    LOCAL CONST Robtarget Tr_meulage_bavure_379 := [[8.9303857421875,-168.09725,77.5905703125],[0.760092273440949,-0.627413460069246,0.107679305140414,-0.130450194418344],[0,0,0,0],[8.999999E+09,8.999999E+09,8.999999E+09,8.999999E+09,8.999999E+09,8.999999E+09]];
    LOCAL CONST Robtarget Tr_meulage_bavure_380 := [[6.36778564453125,-166.2545,77.61740625],[0.757380069640721,-0.624678423253224,0.120981857756658,-0.146682267935255],[0,0,0,0],[8.999999E+09,8.999999E+09,8.999999E+09,8.999999E+09,8.999999E+09,8.999999E+09]];
    LOCAL CONST Robtarget Tr_meulage_bavure_381 := [[0.0211522235870361,-161.8668125,77.659015625],[0.755787418378999,-0.622904489845863,0.128428166406746,-0.155825481944626],[0,0,0,0],[8.999999E+09,8.999999E+09,8.999999E+09,8.999999E+09,8.999999E+09,8.999999E+09]];
    LOCAL CONST Robtarget Tr_meulage_bavure_382 := [[-4.13824365234375,-159.009953125,77.6836484375],[0.75532643398599,-0.622107777939022,0.131008038074695,-0.159062203900237],[0,0,0,0],[8.999999E+09,8.999999E+09,8.999999E+09,8.999999E+09,8.999999E+09,8.999999E+09]];
    LOCAL CONST Robtarget Tr_meulage_bavure_383 := [[-6.49300439453125,-157.311875,77.7089765625],[0.755817096690397,-0.622133912444517,0.129761641555208,-0.157644624766832],[0,0,0,0],[8.999999E+09,8.999999E+09,8.999999E+09,8.999999E+09,8.999999E+09,8.999999E+09]];
    LOCAL CONST Robtarget Tr_meulage_bavure_384 := [[-7.27819287109375,-156.766953125,77.714421875],[0.756985671882866,-0.622757763981476,0.125698769882492,-0.152791620237717],[0,0,0,0],[8.999999E+09,8.999999E+09,8.999999E+09,8.999999E+09,8.999999E+09,8.999999E+09]];
    LOCAL CONST Robtarget Tr_meulage_bavure_385 := [[-7.3110322265625,-156.78715625,77.7085859375],[0.758538176477072,-0.623736548693659,0.119790927466895,-0.14568008219102],[0,0,0,0],[8.999999E+09,8.999999E+09,8.999999E+09,8.999999E+09,8.999999E+09,8.999999E+09]];
    LOCAL CONST Robtarget Tr_meulage_bavure_386 := [[-10.1234833984375,-155.486203125,77.6362265625],[0.760196318256337,-0.624846439022857,0.112999081170998,-0.137476154312211],[0,0,0,0],[8.999999E+09,8.999999E+09,8.999999E+09,8.999999E+09,8.999999E+09,8.999999E+09]];
    LOCAL CONST Robtarget Tr_meulage_bavure_387 := [[-10.6625419921875,-155.202578125,77.6271875],[0.761746908687365,-0.625914144918721,0.106180842065471,-0.129223678457846],[0,0,0,0],[8.999999E+09,8.999999E+09,8.999999E+09,8.999999E+09,8.999999E+09,8.999999E+09]];
    LOCAL CONST Robtarget Tr_meulage_bavure_388 := [[-12.2218876953125,-154.823703125,77.53875],[0.763048486638023,-0.626818658409292,0.100073150713779,-0.121822580072891],[0,0,0,0],[8.999999E+09,8.999999E+09,8.999999E+09,8.999999E+09,8.999999E+09,8.999999E+09]];
    LOCAL CONST Robtarget Tr_meulage_bavure_389 := [[-13.7799794921875,-154.60521875,77.42778125],[0.764015045491845,-0.62749443057358,0.0952699651388726,-0.115997343088844],[0,0,0,0],[8.999999E+09,8.999999E+09,8.999999E+09,8.999999E+09,8.999999E+09,8.999999E+09]];
    LOCAL CONST Robtarget Tr_meulage_bavure_390 := [[-14.96165625,-154.561921875,77.3263515625],[0.764604259131724,-0.627907931444273,0.0922133285385718,-0.112288283390735],[0,0,0,0],[8.999999E+09,8.999999E+09,8.999999E+09,8.999999E+09,8.999999E+09,8.999999E+09]];
    LOCAL CONST Robtarget Tr_meulage_bavure_391 := [[-16.279068359375,-154.44878125,77.222421875],[0.764800293575778,-0.62804670288681,0.0911701159971482,-0.111021889231259],[0,0,0,0],[8.999999E+09,8.999999E+09,8.999999E+09,8.999999E+09,8.999999E+09,8.999999E+09]];
    !
    !Declaration des points de tronconnage

    !
    !Cycle
    LOCAL PROC Cycle()
        !
        Prise;
        !
        Meulage;
        !
        !
        Depose;
        !
    ENDPROC

    !Trajectoire de prise de la pièce
    LOCAL PROC PRISE()

		!
        !Trigger localisation
        LocalisationPieceTable 810 \model:=1;
        !
        !Approche
		MoveJ Reltool(PicKPosition,0,0,-100),V1000,Z0,Tool_Prehenseur1 \Wobj:=Wobj_vision;
		MoveL Reltool(PicKPosition,0,0,-50),V500,Z0,Tool_Prehenseur1 \Wobj:=Wobj_vision;
		MoveL Reltool(PicKPosition,0,0,-10),V200,Z0,Tool_Prehenseur1 \Wobj:=Wobj_vision;
		MoveL PicKPosition,V100,Fine,Tool_Prehenseur1 \Wobj:=Wobj_vision;

        !Fermeture pince
		Gripper_Close;
        !
		MoveL Reltool(PicKPosition,0,0,-100),V500,Z0,Tool_Prehenseur1 \Wobj:=Wobj_vision;

        !Trigger relocalisation
		LocalisationPiecePrehenseur 810 \model:=1,Ref;
        !
        PEO;
        !
    ENDPROC

    !Trajectoire de tronconnage
    LOCAL PROC Tronconnage()
        !
        !StartMotor1();
        !
        ConfJ \Off;
        ConfL \Off;


    ENDPROC


    !Trajectoire de meulage
    LOCAL PROC Meulage()
        !
        !StartMotor2();
        !

        ConfJ \Off;
        ConfL \Off;


        !---------- Meulage zone : 1 ------------

        !Approche PLAN

        Go_to_Meulage_Plan;
		Tool := ToolOffset(Tool_M1_D500_S0 \Z);

        !
        !Approche
        MoveJ Reltool(Tr_meulage_motif_1_0,0,0,-200),V1000,Z0,Tool \Wobj:=Wobj_Part_0;
        MoveL Reltool(Tr_meulage_motif_1_0,0,0,-100),V500,Z0,Tool \Wobj:=Wobj_Part_0;
        MoveL Reltool(Tr_meulage_motif_1_0,0,0,-10),V100,Z0,Tool \Wobj:=Wobj_Part_0;
        !
        !Trajectoire
        Movel Tr_meulage_motif_1_0,VitesseLente,Z0,Tool \Wobj:=Wobj_Part_0;
        Movel Tr_meulage_motif_1_1,VitesseLente,Z0,Tool \Wobj:=Wobj_Part_0;
        Movel Tr_meulage_motif_1_2,VitesseLente,Z0,Tool \Wobj:=Wobj_Part_0;
        Movel Tr_meulage_motif_1_3,VitesseLente,Z0,Tool \Wobj:=Wobj_Part_0;
        Movel Tr_meulage_motif_1_4,VitesseLente,Z0,Tool \Wobj:=Wobj_Part_0;
        Movel Tr_meulage_motif_1_5,VitesseLente,Z0,Tool \Wobj:=Wobj_Part_0;
        Movel Tr_meulage_motif_1_6,VitesseLente,Z0,Tool \Wobj:=Wobj_Part_0;
        Movel Tr_meulage_motif_1_7,VitesseLente,Z0,Tool \Wobj:=Wobj_Part_0;
        Movel Tr_meulage_motif_1_8,VitesseLente,Z0,Tool \Wobj:=Wobj_Part_0;
        Movel Tr_meulage_motif_1_9,VitesseLente,Z0,Tool \Wobj:=Wobj_Part_0;
        Movel Tr_meulage_motif_1_10,VitesseLente,Z0,Tool \Wobj:=Wobj_Part_0;
        Movel Tr_meulage_motif_1_11,VitesseLente,Z0,Tool \Wobj:=Wobj_Part_0;
        Movel Tr_meulage_motif_1_12,VitesseLente,Z0,Tool \Wobj:=Wobj_Part_0;
        Movel Tr_meulage_motif_1_13,VitesseLente,Z0,Tool \Wobj:=Wobj_Part_0;
        Movel Tr_meulage_motif_1_14,VitesseLente,Z0,Tool \Wobj:=Wobj_Part_0;
        Movel Tr_meulage_motif_1_15,VitesseLente,Z0,Tool \Wobj:=Wobj_Part_0;
        Movel Tr_meulage_motif_1_16,VitesseLente,Z0,Tool \Wobj:=Wobj_Part_0;
        Movel Tr_meulage_motif_1_17,VitesseLente,Z0,Tool \Wobj:=Wobj_Part_0;
        Movel Tr_meulage_motif_1_18,VitesseLente,Z0,Tool \Wobj:=Wobj_Part_0;
        Movel Tr_meulage_motif_1_19,VitesseLente,Z0,Tool \Wobj:=Wobj_Part_0;
        Movel Tr_meulage_motif_1_20,VitesseLente,Z0,Tool \Wobj:=Wobj_Part_0;
        Movel Tr_meulage_motif_1_21,VitesseLente,Z0,Tool \Wobj:=Wobj_Part_0;
        Movel Tr_meulage_motif_1_22,VitesseLente,Z0,Tool \Wobj:=Wobj_Part_0;
        Movel Tr_meulage_motif_1_23,VitesseLente,Z0,Tool \Wobj:=Wobj_Part_0;
        Movel Tr_meulage_motif_1_24,VitesseLente,Z0,Tool \Wobj:=Wobj_Part_0;
        Movel Tr_meulage_motif_1_25,VitesseLente,Z0,Tool \Wobj:=Wobj_Part_0;
        Movel Tr_meulage_motif_1_26,VitesseLente,Z0,Tool \Wobj:=Wobj_Part_0;
        Movel Tr_meulage_motif_1_27,VitesseLente,Z0,Tool \Wobj:=Wobj_Part_0;
        Movel Tr_meulage_motif_1_28,VitesseLente,Z0,Tool \Wobj:=Wobj_Part_0;
        Movel Tr_meulage_motif_1_29,VitesseLente,Z0,Tool \Wobj:=Wobj_Part_0;
        Movel Tr_meulage_motif_1_30,VitesseLente,Z0,Tool \Wobj:=Wobj_Part_0;
        Movel Tr_meulage_motif_1_31,VitesseLente,Z0,Tool \Wobj:=Wobj_Part_0;
        Movel Tr_meulage_motif_1_32,VitesseLente,Z0,Tool \Wobj:=Wobj_Part_0;
        Movel Tr_meulage_motif_1_33,VitesseLente,Z0,Tool \Wobj:=Wobj_Part_0;
        Movel Tr_meulage_motif_1_34,VitesseLente,Z0,Tool \Wobj:=Wobj_Part_0;
        Movel Tr_meulage_motif_1_35,VitesseLente,Z0,Tool \Wobj:=Wobj_Part_0;
        Movel Tr_meulage_motif_1_36,VitesseLente,Z0,Tool \Wobj:=Wobj_Part_0;
        Movel Tr_meulage_motif_1_37,VitesseLente,Z0,Tool \Wobj:=Wobj_Part_0;
        Movel Tr_meulage_motif_1_38,VitesseLente,Z0,Tool \Wobj:=Wobj_Part_0;
        Movel Tr_meulage_motif_1_39,VitesseLente,Z0,Tool \Wobj:=Wobj_Part_0;
        Movel Tr_meulage_motif_1_40,VitesseLente,Z0,Tool \Wobj:=Wobj_Part_0;
        Movel Tr_meulage_motif_1_41,VitesseLente,Z0,Tool \Wobj:=Wobj_Part_0;
        Movel Tr_meulage_motif_1_42,VitesseLente,Z0,Tool \Wobj:=Wobj_Part_0;
        Movel Tr_meulage_motif_1_43,VitesseLente,Z0,Tool \Wobj:=Wobj_Part_0;
        Movel Tr_meulage_motif_1_44,VitesseLente,Z0,Tool \Wobj:=Wobj_Part_0;
        Movel Tr_meulage_motif_1_45,VitesseLente,Z0,Tool \Wobj:=Wobj_Part_0;
        Movel Tr_meulage_motif_1_46,VitesseLente,Z0,Tool \Wobj:=Wobj_Part_0;
        Movel Tr_meulage_motif_1_47,VitesseLente,Z0,Tool \Wobj:=Wobj_Part_0;
        Movel Tr_meulage_motif_1_48,VitesseLente,Z0,Tool \Wobj:=Wobj_Part_0;
        Movel Tr_meulage_motif_1_49,VitesseLente,Z0,Tool \Wobj:=Wobj_Part_0;
        Movel Tr_meulage_motif_1_50,VitesseLente,Z0,Tool \Wobj:=Wobj_Part_0;
        Movel Tr_meulage_motif_1_51,VitesseLente,Z0,Tool \Wobj:=Wobj_Part_0;
        Movel Tr_meulage_motif_1_52,VitesseLente,Z0,Tool \Wobj:=Wobj_Part_0;
        Movel Tr_meulage_motif_1_53,VitesseLente,Z0,Tool \Wobj:=Wobj_Part_0;
        Movel Tr_meulage_motif_1_54,VitesseLente,Z0,Tool \Wobj:=Wobj_Part_0;
        Movel Tr_meulage_motif_1_55,VitesseLente,Z0,Tool \Wobj:=Wobj_Part_0;
        Movel Tr_meulage_motif_1_56,VitesseLente,Z0,Tool \Wobj:=Wobj_Part_0;
        Movel Tr_meulage_motif_1_57,VitesseLente,Z0,Tool \Wobj:=Wobj_Part_0;
        Movel Tr_meulage_motif_1_58,VitesseLente,Z0,Tool \Wobj:=Wobj_Part_0;
        Movel Tr_meulage_motif_1_59,VitesseLente,Z0,Tool \Wobj:=Wobj_Part_0;
        Movel Tr_meulage_motif_1_60,VitesseLente,Z0,Tool \Wobj:=Wobj_Part_0;
        Movel Tr_meulage_motif_1_61,VitesseLente,Z0,Tool \Wobj:=Wobj_Part_0;
        Movel Tr_meulage_motif_1_62,VitesseLente,Z0,Tool \Wobj:=Wobj_Part_0;
        Movel Tr_meulage_motif_1_63,VitesseLente,Z0,Tool \Wobj:=Wobj_Part_0;
        Movel Tr_meulage_motif_1_64,VitesseLente,Z0,Tool \Wobj:=Wobj_Part_0;
        Movel Tr_meulage_motif_1_65,VitesseLente,Z0,Tool \Wobj:=Wobj_Part_0;
        Movel Tr_meulage_motif_1_66,VitesseLente,Z0,Tool \Wobj:=Wobj_Part_0;
        Movel Tr_meulage_motif_1_67,VitesseLente,Z0,Tool \Wobj:=Wobj_Part_0;
        Movel Tr_meulage_motif_1_68,VitesseLente,Z0,Tool \Wobj:=Wobj_Part_0;
        Movel Tr_meulage_motif_1_69,VitesseLente,Z0,Tool \Wobj:=Wobj_Part_0;
        Movel Tr_meulage_motif_1_70,VitesseLente,Z0,Tool \Wobj:=Wobj_Part_0;
        Movel Tr_meulage_motif_1_71,VitesseLente,Z0,Tool \Wobj:=Wobj_Part_0;
        Movel Tr_meulage_motif_1_72,VitesseLente,Z0,Tool \Wobj:=Wobj_Part_0;
        Movel Tr_meulage_motif_1_73,VitesseLente,Z0,Tool \Wobj:=Wobj_Part_0;
        Movel Tr_meulage_motif_1_74,VitesseLente,Z0,Tool \Wobj:=Wobj_Part_0;
        Movel Tr_meulage_motif_1_75,VitesseLente,Z0,Tool \Wobj:=Wobj_Part_0;
        Movel Tr_meulage_motif_1_76,VitesseLente,Z0,Tool \Wobj:=Wobj_Part_0;
        Movel Tr_meulage_motif_1_77,VitesseLente,Z0,Tool \Wobj:=Wobj_Part_0;
        Movel Tr_meulage_motif_1_78,VitesseLente,Z0,Tool \Wobj:=Wobj_Part_0;
        Movel Tr_meulage_motif_1_79,VitesseLente,Z0,Tool \Wobj:=Wobj_Part_0;
        Movel Tr_meulage_motif_1_80,VitesseLente,Z0,Tool \Wobj:=Wobj_Part_0;
        Movel Tr_meulage_motif_1_81,VitesseLente,Z0,Tool \Wobj:=Wobj_Part_0;
        Movel Tr_meulage_motif_1_82,VitesseLente,Z0,Tool \Wobj:=Wobj_Part_0;
        Movel Tr_meulage_motif_1_83,VitesseLente,Z0,Tool \Wobj:=Wobj_Part_0;
        Movel Tr_meulage_motif_1_84,VitesseLente,Z0,Tool \Wobj:=Wobj_Part_0;
        Movel Tr_meulage_motif_1_85,VitesseLente,Z0,Tool \Wobj:=Wobj_Part_0;
        Movel Tr_meulage_motif_1_86,VitesseLente,Z0,Tool \Wobj:=Wobj_Part_0;
        Movel Tr_meulage_motif_1_87,VitesseLente,Z0,Tool \Wobj:=Wobj_Part_0;
        Movel Tr_meulage_motif_1_88,VitesseLente,Z0,Tool \Wobj:=Wobj_Part_0;
        Movel Tr_meulage_motif_1_89,VitesseLente,Z0,Tool \Wobj:=Wobj_Part_0;
        Movel Tr_meulage_motif_1_90,VitesseLente,Z0,Tool \Wobj:=Wobj_Part_0;
        Movel Tr_meulage_motif_1_91,VitesseLente,Z0,Tool \Wobj:=Wobj_Part_0;
        Movel Tr_meulage_motif_1_92,VitesseLente,Z0,Tool \Wobj:=Wobj_Part_0;
        Movel Tr_meulage_motif_1_93,VitesseLente,Z0,Tool \Wobj:=Wobj_Part_0;
        Movel Tr_meulage_motif_1_94,VitesseLente,Z0,Tool \Wobj:=Wobj_Part_0;
        Movel Tr_meulage_motif_1_95,VitesseLente,Z0,Tool \Wobj:=Wobj_Part_0;
        Movel Tr_meulage_motif_1_96,VitesseLente,Z0,Tool \Wobj:=Wobj_Part_0;
        Movel Tr_meulage_motif_1_97,VitesseLente,Z0,Tool \Wobj:=Wobj_Part_0;
        Movel Tr_meulage_motif_1_98,VitesseLente,Z0,Tool \Wobj:=Wobj_Part_0;
        Movel Tr_meulage_motif_1_99,VitesseLente,Z0,Tool \Wobj:=Wobj_Part_0;
        Movel Tr_meulage_motif_1_100,VitesseLente,Z0,Tool \Wobj:=Wobj_Part_0;
        Movel Tr_meulage_motif_1_101,VitesseLente,Z0,Tool \Wobj:=Wobj_Part_0;
        Movel Tr_meulage_motif_1_102,VitesseLente,Z0,Tool \Wobj:=Wobj_Part_0;
        Movel Tr_meulage_motif_1_103,VitesseLente,Z0,Tool \Wobj:=Wobj_Part_0;
        Movel Tr_meulage_motif_1_104,VitesseLente,Z0,Tool \Wobj:=Wobj_Part_0;
        Movel Tr_meulage_motif_1_105,VitesseLente,Z0,Tool \Wobj:=Wobj_Part_0;
        Movel Tr_meulage_motif_1_106,VitesseLente,Z0,Tool \Wobj:=Wobj_Part_0;
        Movel Tr_meulage_motif_1_107,VitesseLente,Z0,Tool \Wobj:=Wobj_Part_0;
        Movel Tr_meulage_motif_1_108,VitesseLente,Z0,Tool \Wobj:=Wobj_Part_0;
        Movel Tr_meulage_motif_1_109,VitesseLente,Z0,Tool \Wobj:=Wobj_Part_0;
        Movel Tr_meulage_motif_1_110,VitesseLente,Z0,Tool \Wobj:=Wobj_Part_0;
        Movel Tr_meulage_motif_1_111,VitesseLente,Z0,Tool \Wobj:=Wobj_Part_0;
        Movel Tr_meulage_motif_1_112,VitesseLente,Z0,Tool \Wobj:=Wobj_Part_0;
        Movel Tr_meulage_motif_1_113,VitesseLente,Z0,Tool \Wobj:=Wobj_Part_0;
        Movel Tr_meulage_motif_1_114,VitesseLente,Z0,Tool \Wobj:=Wobj_Part_0;
        Movel Tr_meulage_motif_1_115,VitesseLente,Z0,Tool \Wobj:=Wobj_Part_0;
        Movel Tr_meulage_motif_1_116,VitesseLente,Z0,Tool \Wobj:=Wobj_Part_0;
        Movel Tr_meulage_motif_1_117,VitesseLente,Z0,Tool \Wobj:=Wobj_Part_0;
        Movel Tr_meulage_motif_1_118,VitesseLente,Z0,Tool \Wobj:=Wobj_Part_0;
        Movel Tr_meulage_motif_1_119,VitesseLente,Z0,Tool \Wobj:=Wobj_Part_0;
        Movel Tr_meulage_motif_1_120,VitesseLente,Z0,Tool \Wobj:=Wobj_Part_0;
        Movel Tr_meulage_motif_1_121,VitesseLente,Z0,Tool \Wobj:=Wobj_Part_0;
        Movel Tr_meulage_motif_1_122,VitesseLente,Z0,Tool \Wobj:=Wobj_Part_0;
        Movel Tr_meulage_motif_1_123,VitesseLente,Z0,Tool \Wobj:=Wobj_Part_0;
        Movel Tr_meulage_motif_1_124,VitesseLente,Z0,Tool \Wobj:=Wobj_Part_0;
        Movel Tr_meulage_motif_1_125,VitesseLente,Z0,Tool \Wobj:=Wobj_Part_0;
        Movel Tr_meulage_motif_1_126,VitesseLente,Z0,Tool \Wobj:=Wobj_Part_0;
        Movel Tr_meulage_motif_1_127,VitesseLente,Z0,Tool \Wobj:=Wobj_Part_0;
        Movel Tr_meulage_motif_1_128,VitesseLente,Z0,Tool \Wobj:=Wobj_Part_0;
        Movel Tr_meulage_motif_1_129,VitesseLente,Z0,Tool \Wobj:=Wobj_Part_0;
        Movel Tr_meulage_motif_1_130,VitesseLente,Z0,Tool \Wobj:=Wobj_Part_0;
        Movel Tr_meulage_motif_1_131,VitesseLente,Z0,Tool \Wobj:=Wobj_Part_0;
        Movel Tr_meulage_motif_1_132,VitesseLente,Z0,Tool \Wobj:=Wobj_Part_0;
        Movel Tr_meulage_motif_1_133,VitesseLente,Z0,Tool \Wobj:=Wobj_Part_0;
        Movel Tr_meulage_motif_1_134,VitesseLente,Z0,Tool \Wobj:=Wobj_Part_0;
        Movel Tr_meulage_motif_1_135,VitesseLente,Z0,Tool \Wobj:=Wobj_Part_0;
        Movel Tr_meulage_motif_1_136,VitesseLente,Z0,Tool \Wobj:=Wobj_Part_0;
        Movel Tr_meulage_motif_1_137,VitesseLente,Z0,Tool \Wobj:=Wobj_Part_0;
        Movel Tr_meulage_motif_1_138,VitesseLente,Z0,Tool \Wobj:=Wobj_Part_0;
        Movel Tr_meulage_motif_1_139,VitesseLente,Z0,Tool \Wobj:=Wobj_Part_0;
        Movel Tr_meulage_motif_1_140,VitesseLente,Z0,Tool \Wobj:=Wobj_Part_0;
        Movel Tr_meulage_motif_1_141,VitesseLente,Z0,Tool \Wobj:=Wobj_Part_0;
        Movel Tr_meulage_motif_1_142,VitesseLente,Z0,Tool \Wobj:=Wobj_Part_0;
        Movel Tr_meulage_motif_1_143,VitesseLente,Z0,Tool \Wobj:=Wobj_Part_0;
        Movel Tr_meulage_motif_1_144,VitesseLente,Z0,Tool \Wobj:=Wobj_Part_0;
        Movel Tr_meulage_motif_1_145,VitesseLente,Z0,Tool \Wobj:=Wobj_Part_0;
        Movel Tr_meulage_motif_1_146,VitesseLente,Z0,Tool \Wobj:=Wobj_Part_0;
        Movel Tr_meulage_motif_1_147,VitesseLente,Z0,Tool \Wobj:=Wobj_Part_0;
        Movel Tr_meulage_motif_1_148,VitesseLente,Z0,Tool \Wobj:=Wobj_Part_0;
        Movel Tr_meulage_motif_1_149,VitesseLente,Z0,Tool \Wobj:=Wobj_Part_0;
        Movel Tr_meulage_motif_1_150,VitesseLente,Z0,Tool \Wobj:=Wobj_Part_0;
        Movel Tr_meulage_motif_1_151,VitesseLente,Z0,Tool \Wobj:=Wobj_Part_0;
        Movel Tr_meulage_motif_1_152,VitesseLente,Z0,Tool \Wobj:=Wobj_Part_0;
        Movel Tr_meulage_motif_1_153,VitesseLente,Z0,Tool \Wobj:=Wobj_Part_0;
        Movel Tr_meulage_motif_1_154,VitesseLente,Z0,Tool \Wobj:=Wobj_Part_0;
        Movel Tr_meulage_motif_1_155,VitesseLente,Z0,Tool \Wobj:=Wobj_Part_0;
        Movel Tr_meulage_motif_1_156,VitesseLente,Z0,Tool \Wobj:=Wobj_Part_0;
        Movel Tr_meulage_motif_1_157,VitesseLente,Z0,Tool \Wobj:=Wobj_Part_0;
        Movel Tr_meulage_motif_1_158,VitesseLente,Z0,Tool \Wobj:=Wobj_Part_0;
        Movel Tr_meulage_motif_1_159,VitesseLente,Z0,Tool \Wobj:=Wobj_Part_0;
        Movel Tr_meulage_motif_1_160,VitesseLente,Z0,Tool \Wobj:=Wobj_Part_0;
        Movel Tr_meulage_motif_1_161,VitesseLente,Z0,Tool \Wobj:=Wobj_Part_0;
        Movel Tr_meulage_motif_1_162,VitesseLente,Z0,Tool \Wobj:=Wobj_Part_0;
        Movel Tr_meulage_motif_1_163,VitesseLente,Z0,Tool \Wobj:=Wobj_Part_0;
        Movel Tr_meulage_motif_1_164,VitesseLente,Z0,Tool \Wobj:=Wobj_Part_0;
        Movel Tr_meulage_motif_1_165,VitesseLente,Z0,Tool \Wobj:=Wobj_Part_0;
        Movel Tr_meulage_motif_1_166,VitesseLente,Z0,Tool \Wobj:=Wobj_Part_0;
        Movel Tr_meulage_motif_1_167,VitesseLente,Z0,Tool \Wobj:=Wobj_Part_0;
        Movel Tr_meulage_motif_1_168,VitesseLente,Z0,Tool \Wobj:=Wobj_Part_0;
        Movel Tr_meulage_motif_1_169,VitesseLente,Z0,Tool \Wobj:=Wobj_Part_0;
        Movel Tr_meulage_motif_1_170,VitesseLente,Z0,Tool \Wobj:=Wobj_Part_0;
        Movel Tr_meulage_motif_1_171,VitesseLente,Z0,Tool \Wobj:=Wobj_Part_0;
        Movel Tr_meulage_motif_1_172,VitesseLente,Z0,Tool \Wobj:=Wobj_Part_0;
        Movel Tr_meulage_motif_1_173,VitesseLente,Z0,Tool \Wobj:=Wobj_Part_0;
        Movel Tr_meulage_motif_1_174,VitesseLente,Z0,Tool \Wobj:=Wobj_Part_0;
        Movel Tr_meulage_motif_1_175,VitesseLente,Z0,Tool \Wobj:=Wobj_Part_0;
        Movel Tr_meulage_motif_1_176,VitesseLente,Z0,Tool \Wobj:=Wobj_Part_0;
        Movel Tr_meulage_motif_1_177,VitesseLente,Z0,Tool \Wobj:=Wobj_Part_0;
        Movel Tr_meulage_motif_1_178,VitesseLente,Z0,Tool \Wobj:=Wobj_Part_0;
        Movel Tr_meulage_motif_1_179,VitesseLente,Z0,Tool \Wobj:=Wobj_Part_0;
        Movel Tr_meulage_motif_1_180,VitesseLente,Z0,Tool \Wobj:=Wobj_Part_0;
        Movel Tr_meulage_motif_1_181,VitesseLente,Z0,Tool \Wobj:=Wobj_Part_0;
        Movel Tr_meulage_motif_1_182,VitesseLente,Z0,Tool \Wobj:=Wobj_Part_0;
        Movel Tr_meulage_motif_1_183,VitesseLente,Z0,Tool \Wobj:=Wobj_Part_0;
        Movel Tr_meulage_motif_1_184,VitesseLente,Z0,Tool \Wobj:=Wobj_Part_0;
        Movel Tr_meulage_motif_1_185,VitesseLente,Z0,Tool \Wobj:=Wobj_Part_0;
        Movel Tr_meulage_motif_1_186,VitesseLente,Z0,Tool \Wobj:=Wobj_Part_0;
        Movel Tr_meulage_motif_1_187,VitesseLente,Z0,Tool \Wobj:=Wobj_Part_0;
        Movel Tr_meulage_motif_1_188,VitesseLente,Z0,Tool \Wobj:=Wobj_Part_0;
        Movel Tr_meulage_motif_1_189,VitesseLente,Z0,Tool \Wobj:=Wobj_Part_0;
        Movel Tr_meulage_motif_1_190,VitesseLente,Z0,Tool \Wobj:=Wobj_Part_0;
        Movel Tr_meulage_motif_1_191,VitesseLente,Z0,Tool \Wobj:=Wobj_Part_0;
        Movel Tr_meulage_motif_1_192,VitesseLente,Z0,Tool \Wobj:=Wobj_Part_0;
        Movel Tr_meulage_motif_1_193,VitesseLente,Z0,Tool \Wobj:=Wobj_Part_0;
        Movel Tr_meulage_motif_1_194,VitesseLente,Z0,Tool \Wobj:=Wobj_Part_0;
        Movel Tr_meulage_motif_1_195,VitesseLente,Z0,Tool \Wobj:=Wobj_Part_0;
        Movel Tr_meulage_motif_1_196,VitesseLente,Z0,Tool \Wobj:=Wobj_Part_0;
        Movel Tr_meulage_motif_1_197,VitesseLente,Z0,Tool \Wobj:=Wobj_Part_0;
        Movel Tr_meulage_motif_1_198,VitesseLente,Z0,Tool \Wobj:=Wobj_Part_0;
        Movel Tr_meulage_motif_1_199,VitesseLente,Z0,Tool \Wobj:=Wobj_Part_0;
        Movel Tr_meulage_motif_1_200,VitesseLente,Z0,Tool \Wobj:=Wobj_Part_0;
        Movel Tr_meulage_motif_1_201,VitesseLente,Z0,Tool \Wobj:=Wobj_Part_0;
        Movel Tr_meulage_motif_1_202,VitesseLente,Z0,Tool \Wobj:=Wobj_Part_0;
        Movel Tr_meulage_motif_1_203,VitesseLente,Z0,Tool \Wobj:=Wobj_Part_0;
        Movel Tr_meulage_motif_1_204,VitesseLente,Z0,Tool \Wobj:=Wobj_Part_0;
        Movel Tr_meulage_motif_1_205,VitesseLente,Z0,Tool \Wobj:=Wobj_Part_0;
        Movel Tr_meulage_motif_1_206,VitesseLente,Z0,Tool \Wobj:=Wobj_Part_0;
        Movel Tr_meulage_motif_1_207,VitesseLente,Z0,Tool \Wobj:=Wobj_Part_0;
        Movel Tr_meulage_motif_1_208,VitesseLente,Z0,Tool \Wobj:=Wobj_Part_0;
        Movel Tr_meulage_motif_1_209,VitesseLente,Z0,Tool \Wobj:=Wobj_Part_0;
        Movel Tr_meulage_motif_1_210,VitesseLente,Z0,Tool \Wobj:=Wobj_Part_0;
        Movel Tr_meulage_motif_1_211,VitesseLente,Z0,Tool \Wobj:=Wobj_Part_0;
        Movel Tr_meulage_motif_1_212,VitesseLente,Z0,Tool \Wobj:=Wobj_Part_0;
        Movel Tr_meulage_motif_1_213,VitesseLente,Z0,Tool \Wobj:=Wobj_Part_0;
        Movel Tr_meulage_motif_1_214,VitesseLente,Z0,Tool \Wobj:=Wobj_Part_0;
        Movel Tr_meulage_motif_1_215,VitesseLente,Z0,Tool \Wobj:=Wobj_Part_0;
        Movel Tr_meulage_motif_1_216,VitesseLente,Z0,Tool \Wobj:=Wobj_Part_0;
        Movel Tr_meulage_motif_1_217,VitesseLente,Z0,Tool \Wobj:=Wobj_Part_0;
        Movel Tr_meulage_motif_1_218,VitesseLente,Z0,Tool \Wobj:=Wobj_Part_0;
        Movel Tr_meulage_motif_1_219,VitesseLente,Z0,Tool \Wobj:=Wobj_Part_0;
        Movel Tr_meulage_motif_1_220,VitesseLente,Z0,Tool \Wobj:=Wobj_Part_0;
        Movel Tr_meulage_motif_1_221,VitesseLente,Z0,Tool \Wobj:=Wobj_Part_0;
        Movel Tr_meulage_motif_1_222,VitesseLente,Z0,Tool \Wobj:=Wobj_Part_0;
        Movel Tr_meulage_motif_1_223,VitesseLente,Z0,Tool \Wobj:=Wobj_Part_0;
        Movel Tr_meulage_motif_1_224,VitesseLente,Z0,Tool \Wobj:=Wobj_Part_0;
        Movel Tr_meulage_motif_1_225,VitesseLente,Z0,Tool \Wobj:=Wobj_Part_0;
        Movel Tr_meulage_motif_1_226,VitesseLente,Z0,Tool \Wobj:=Wobj_Part_0;
        Movel Tr_meulage_motif_1_227,VitesseLente,Z0,Tool \Wobj:=Wobj_Part_0;
        Movel Tr_meulage_motif_1_228,VitesseLente,Z0,Tool \Wobj:=Wobj_Part_0;
        Movel Tr_meulage_motif_1_229,VitesseLente,Z0,Tool \Wobj:=Wobj_Part_0;
        Movel Tr_meulage_motif_1_230,VitesseLente,Z0,Tool \Wobj:=Wobj_Part_0;
        Movel Tr_meulage_motif_1_231,VitesseLente,Z0,Tool \Wobj:=Wobj_Part_0;
        Movel Tr_meulage_motif_1_232,VitesseLente,Z0,Tool \Wobj:=Wobj_Part_0;
        Movel Tr_meulage_motif_1_233,VitesseLente,Z0,Tool \Wobj:=Wobj_Part_0;
        Movel Tr_meulage_motif_1_234,VitesseLente,Z0,Tool \Wobj:=Wobj_Part_0;
        Movel Tr_meulage_motif_1_235,VitesseLente,Z0,Tool \Wobj:=Wobj_Part_0;
        Movel Tr_meulage_motif_1_236,VitesseLente,Z0,Tool \Wobj:=Wobj_Part_0;
        Movel Tr_meulage_motif_1_237,VitesseLente,Z0,Tool \Wobj:=Wobj_Part_0;
        Movel Tr_meulage_motif_1_238,VitesseLente,Z0,Tool \Wobj:=Wobj_Part_0;
        Movel Tr_meulage_motif_1_239,VitesseLente,Z0,Tool \Wobj:=Wobj_Part_0;
        Movel Tr_meulage_motif_1_240,VitesseLente,Z0,Tool \Wobj:=Wobj_Part_0;
        Movel Tr_meulage_motif_1_241,VitesseLente,Z0,Tool \Wobj:=Wobj_Part_0;
        Movel Tr_meulage_motif_1_242,VitesseLente,Z0,Tool \Wobj:=Wobj_Part_0;
        Movel Tr_meulage_motif_1_243,VitesseLente,Z0,Tool \Wobj:=Wobj_Part_0;
        Movel Tr_meulage_motif_1_244,VitesseLente,Z0,Tool \Wobj:=Wobj_Part_0;
        Movel Tr_meulage_motif_1_245,VitesseLente,Z0,Tool \Wobj:=Wobj_Part_0;
        Movel Tr_meulage_motif_1_246,VitesseLente,Z0,Tool \Wobj:=Wobj_Part_0;
        Movel Tr_meulage_motif_1_247,VitesseLente,Z0,Tool \Wobj:=Wobj_Part_0;
        Movel Tr_meulage_motif_1_248,VitesseLente,Z0,Tool \Wobj:=Wobj_Part_0;
        Movel Tr_meulage_motif_1_249,VitesseLente,Z0,Tool \Wobj:=Wobj_Part_0;
        Movel Tr_meulage_motif_1_250,VitesseLente,Z0,Tool \Wobj:=Wobj_Part_0;
        Movel Tr_meulage_motif_1_251,VitesseLente,Z0,Tool \Wobj:=Wobj_Part_0;
        Movel Tr_meulage_motif_1_252,VitesseLente,Z0,Tool \Wobj:=Wobj_Part_0;
        Movel Tr_meulage_motif_1_253,VitesseLente,Z0,Tool \Wobj:=Wobj_Part_0;
        Movel Tr_meulage_motif_1_254,VitesseLente,Z0,Tool \Wobj:=Wobj_Part_0;
        Movel Tr_meulage_motif_1_255,VitesseLente,Z0,Tool \Wobj:=Wobj_Part_0;
        Movel Tr_meulage_motif_1_256,VitesseLente,Z0,Tool \Wobj:=Wobj_Part_0;
        Movel Tr_meulage_motif_1_257,VitesseLente,Z0,Tool \Wobj:=Wobj_Part_0;
        Movel Tr_meulage_motif_1_258,VitesseLente,Z0,Tool \Wobj:=Wobj_Part_0;
        Movel Tr_meulage_motif_1_259,VitesseLente,Z0,Tool \Wobj:=Wobj_Part_0;
        Movel Tr_meulage_motif_1_260,VitesseLente,Z0,Tool \Wobj:=Wobj_Part_0;
        Movel Tr_meulage_motif_1_261,VitesseLente,Z0,Tool \Wobj:=Wobj_Part_0;
        Movel Tr_meulage_motif_1_262,VitesseLente,Z0,Tool \Wobj:=Wobj_Part_0;
        Movel Tr_meulage_motif_1_263,VitesseLente,Z0,Tool \Wobj:=Wobj_Part_0;
        Movel Tr_meulage_motif_1_264,VitesseLente,Z0,Tool \Wobj:=Wobj_Part_0;
        Movel Tr_meulage_motif_1_265,VitesseLente,Z0,Tool \Wobj:=Wobj_Part_0;
        Movel Tr_meulage_motif_1_266,VitesseLente,Z0,Tool \Wobj:=Wobj_Part_0;
        Movel Tr_meulage_motif_1_267,VitesseLente,Z0,Tool \Wobj:=Wobj_Part_0;
        Movel Tr_meulage_motif_1_268,VitesseLente,Z0,Tool \Wobj:=Wobj_Part_0;
        Movel Tr_meulage_motif_1_269,VitesseLente,Z0,Tool \Wobj:=Wobj_Part_0;
        Movel Tr_meulage_motif_1_270,VitesseLente,Z0,Tool \Wobj:=Wobj_Part_0;
        Movel Tr_meulage_motif_1_271,VitesseLente,Z0,Tool \Wobj:=Wobj_Part_0;
        Movel Tr_meulage_motif_1_272,VitesseLente,Z0,Tool \Wobj:=Wobj_Part_0;
        Movel Tr_meulage_motif_1_273,VitesseLente,Z0,Tool \Wobj:=Wobj_Part_0;
        Movel Tr_meulage_motif_1_274,VitesseLente,Z0,Tool \Wobj:=Wobj_Part_0;
        Movel Tr_meulage_motif_1_275,VitesseLente,Z0,Tool \Wobj:=Wobj_Part_0;
        Movel Tr_meulage_motif_1_276,VitesseLente,Z0,Tool \Wobj:=Wobj_Part_0;
        Movel Tr_meulage_motif_1_277,VitesseLente,Z0,Tool \Wobj:=Wobj_Part_0;
        Movel Tr_meulage_motif_1_278,VitesseLente,Z0,Tool \Wobj:=Wobj_Part_0;
        Movel Tr_meulage_motif_1_279,VitesseLente,Z0,Tool \Wobj:=Wobj_Part_0;
        Movel Tr_meulage_motif_1_280,VitesseLente,Z0,Tool \Wobj:=Wobj_Part_0;
        Movel Tr_meulage_motif_1_281,VitesseLente,Z0,Tool \Wobj:=Wobj_Part_0;
        Movel Tr_meulage_motif_1_282,VitesseLente,Z0,Tool \Wobj:=Wobj_Part_0;
        Movel Tr_meulage_motif_1_283,VitesseLente,Z0,Tool \Wobj:=Wobj_Part_0;
        Movel Tr_meulage_motif_1_284,VitesseLente,Z0,Tool \Wobj:=Wobj_Part_0;
        Movel Tr_meulage_motif_1_285,VitesseLente,Z0,Tool \Wobj:=Wobj_Part_0;
        Movel Tr_meulage_motif_1_286,VitesseLente,Z0,Tool \Wobj:=Wobj_Part_0;
        Movel Tr_meulage_motif_1_287,VitesseLente,Z0,Tool \Wobj:=Wobj_Part_0;
        Movel Tr_meulage_motif_1_288,VitesseLente,Z0,Tool \Wobj:=Wobj_Part_0;
        Movel Tr_meulage_motif_1_289,VitesseLente,Z0,Tool \Wobj:=Wobj_Part_0;
        Movel Tr_meulage_motif_1_290,VitesseLente,Z0,Tool \Wobj:=Wobj_Part_0;
        Movel Tr_meulage_motif_1_291,VitesseLente,Z0,Tool \Wobj:=Wobj_Part_0;
        Movel Tr_meulage_motif_1_292,VitesseLente,Z0,Tool \Wobj:=Wobj_Part_0;
        Movel Tr_meulage_motif_1_293,VitesseLente,Z0,Tool \Wobj:=Wobj_Part_0;
        Movel Tr_meulage_motif_1_294,VitesseLente,Z0,Tool \Wobj:=Wobj_Part_0;
        !
        !Degagement
        MoveL Reltool(Tr_meulage_motif_1_294,0,0,-10),V100,Z0,Tool \Wobj:=Wobj_Part_0;
        MoveL Reltool(Tr_meulage_motif_1_294,0,0,-100),V500,Z0,Tool \Wobj:=Wobj_Part_0;
        MoveJ Reltool(Tr_meulage_motif_1_294,0,0,-200),V1000,Z0,Tool \Wobj:=Wobj_Part_0;


        Go_to_Meulage_Plan;
        !
        !

        !---------- Meulage zone : 2 ------------

        !Approche PLAN

        Go_to_Meulage_Plan;
		Tool := ToolOffset(Tool_M1_D500_S0 \Z);

        !
        !Approche
        MoveJ Reltool(Tr_meulage_bavure_0,0,0,-200),V1000,Z0,Tool \Wobj:=Wobj_Part_0;
        MoveL Reltool(Tr_meulage_bavure_0,0,0,-100),V500,Z0,Tool \Wobj:=Wobj_Part_0;
        MoveL Reltool(Tr_meulage_bavure_0,0,0,-10),V100,Z0,Tool \Wobj:=Wobj_Part_0;
        !
        !Trajectoire
        Movel Tr_meulage_bavure_0,VitesseRapide,Z0,Tool \Wobj:=Wobj_Part_0;
        Movel Tr_meulage_bavure_1,VitesseRapide,Z0,Tool \Wobj:=Wobj_Part_0;
        Movel Tr_meulage_bavure_2,VitesseRapide,Z0,Tool \Wobj:=Wobj_Part_0;
        Movel Tr_meulage_bavure_3,VitesseRapide,Z0,Tool \Wobj:=Wobj_Part_0;
        Movel Tr_meulage_bavure_4,VitesseRapide,Z0,Tool \Wobj:=Wobj_Part_0;
        Movel Tr_meulage_bavure_5,VitesseRapide,Z0,Tool \Wobj:=Wobj_Part_0;
        Movel Tr_meulage_bavure_6,VitesseRapide,Z0,Tool \Wobj:=Wobj_Part_0;
        Movel Tr_meulage_bavure_7,VitesseRapide,Z0,Tool \Wobj:=Wobj_Part_0;
        Movel Tr_meulage_bavure_8,VitesseRapide,Z0,Tool \Wobj:=Wobj_Part_0;
        Movel Tr_meulage_bavure_9,VitesseRapide,Z0,Tool \Wobj:=Wobj_Part_0;
        Movel Tr_meulage_bavure_10,VitesseRapide,Z0,Tool \Wobj:=Wobj_Part_0;
        Movel Tr_meulage_bavure_11,VitesseRapide,Z0,Tool \Wobj:=Wobj_Part_0;
        Movel Tr_meulage_bavure_12,VitesseRapide,Z0,Tool \Wobj:=Wobj_Part_0;
        Movel Tr_meulage_bavure_13,VitesseRapide,Z0,Tool \Wobj:=Wobj_Part_0;
        Movel Tr_meulage_bavure_14,VitesseRapide,Z0,Tool \Wobj:=Wobj_Part_0;
        Movel Tr_meulage_bavure_15,VitesseRapide,Z0,Tool \Wobj:=Wobj_Part_0;
        Movel Tr_meulage_bavure_16,VitesseRapide,Z0,Tool \Wobj:=Wobj_Part_0;
        Movel Tr_meulage_bavure_17,VitesseRapide,Z0,Tool \Wobj:=Wobj_Part_0;
        Movel Tr_meulage_bavure_18,VitesseRapide,Z0,Tool \Wobj:=Wobj_Part_0;
        Movel Tr_meulage_bavure_19,VitesseRapide,Z0,Tool \Wobj:=Wobj_Part_0;
        Movel Tr_meulage_bavure_20,VitesseRapide,Z0,Tool \Wobj:=Wobj_Part_0;
        Movel Tr_meulage_bavure_21,VitesseRapide,Z0,Tool \Wobj:=Wobj_Part_0;
        Movel Tr_meulage_bavure_22,VitesseRapide,Z0,Tool \Wobj:=Wobj_Part_0;
        Movel Tr_meulage_bavure_23,VitesseRapide,Z0,Tool \Wobj:=Wobj_Part_0;
        Movel Tr_meulage_bavure_24,VitesseRapide,Z0,Tool \Wobj:=Wobj_Part_0;
        Movel Tr_meulage_bavure_25,VitesseRapide,Z0,Tool \Wobj:=Wobj_Part_0;
        Movel Tr_meulage_bavure_26,VitesseRapide,Z0,Tool \Wobj:=Wobj_Part_0;
        Movel Tr_meulage_bavure_27,VitesseRapide,Z0,Tool \Wobj:=Wobj_Part_0;
        Movel Tr_meulage_bavure_28,VitesseRapide,Z0,Tool \Wobj:=Wobj_Part_0;
        Movel Tr_meulage_bavure_29,VitesseRapide,Z0,Tool \Wobj:=Wobj_Part_0;
        Movel Tr_meulage_bavure_30,VitesseRapide,Z0,Tool \Wobj:=Wobj_Part_0;
        Movel Tr_meulage_bavure_31,VitesseRapide,Z0,Tool \Wobj:=Wobj_Part_0;
        Movel Tr_meulage_bavure_32,VitesseRapide,Z0,Tool \Wobj:=Wobj_Part_0;
        Movel Tr_meulage_bavure_33,VitesseRapide,Z0,Tool \Wobj:=Wobj_Part_0;
        Movel Tr_meulage_bavure_34,VitesseRapide,Z0,Tool \Wobj:=Wobj_Part_0;
        Movel Tr_meulage_bavure_35,VitesseRapide,Z0,Tool \Wobj:=Wobj_Part_0;
        Movel Tr_meulage_bavure_36,VitesseRapide,Z0,Tool \Wobj:=Wobj_Part_0;
        Movel Tr_meulage_bavure_37,VitesseRapide,Z0,Tool \Wobj:=Wobj_Part_0;
        Movel Tr_meulage_bavure_38,VitesseRapide,Z0,Tool \Wobj:=Wobj_Part_0;
        Movel Tr_meulage_bavure_39,VitesseRapide,Z0,Tool \Wobj:=Wobj_Part_0;
        Movel Tr_meulage_bavure_40,VitesseRapide,Z0,Tool \Wobj:=Wobj_Part_0;
        Movel Tr_meulage_bavure_41,VitesseRapide,Z0,Tool \Wobj:=Wobj_Part_0;
        Movel Tr_meulage_bavure_42,VitesseRapide,Z0,Tool \Wobj:=Wobj_Part_0;
        Movel Tr_meulage_bavure_43,VitesseRapide,Z0,Tool \Wobj:=Wobj_Part_0;
        Movel Tr_meulage_bavure_44,VitesseRapide,Z0,Tool \Wobj:=Wobj_Part_0;
        Movel Tr_meulage_bavure_45,VitesseRapide,Z0,Tool \Wobj:=Wobj_Part_0;
        Movel Tr_meulage_bavure_46,VitesseRapide,Z0,Tool \Wobj:=Wobj_Part_0;
        Movel Tr_meulage_bavure_47,VitesseRapide,Z0,Tool \Wobj:=Wobj_Part_0;
        Movel Tr_meulage_bavure_48,VitesseRapide,Z0,Tool \Wobj:=Wobj_Part_0;
        Movel Tr_meulage_bavure_49,VitesseRapide,Z0,Tool \Wobj:=Wobj_Part_0;
        Movel Tr_meulage_bavure_50,VitesseRapide,Z0,Tool \Wobj:=Wobj_Part_0;
        Movel Tr_meulage_bavure_51,VitesseRapide,Z0,Tool \Wobj:=Wobj_Part_0;
        Movel Tr_meulage_bavure_52,VitesseRapide,Z0,Tool \Wobj:=Wobj_Part_0;
        Movel Tr_meulage_bavure_53,VitesseRapide,Z0,Tool \Wobj:=Wobj_Part_0;
        Movel Tr_meulage_bavure_54,VitesseRapide,Z0,Tool \Wobj:=Wobj_Part_0;
        Movel Tr_meulage_bavure_55,VitesseRapide,Z0,Tool \Wobj:=Wobj_Part_0;
        Movel Tr_meulage_bavure_56,VitesseRapide,Z0,Tool \Wobj:=Wobj_Part_0;
        Movel Tr_meulage_bavure_57,VitesseRapide,Z0,Tool \Wobj:=Wobj_Part_0;
        Movel Tr_meulage_bavure_58,VitesseRapide,Z0,Tool \Wobj:=Wobj_Part_0;
        Movel Tr_meulage_bavure_59,VitesseRapide,Z0,Tool \Wobj:=Wobj_Part_0;
        Movel Tr_meulage_bavure_60,VitesseRapide,Z0,Tool \Wobj:=Wobj_Part_0;
        Movel Tr_meulage_bavure_61,VitesseRapide,Z0,Tool \Wobj:=Wobj_Part_0;
        Movel Tr_meulage_bavure_62,VitesseRapide,Z0,Tool \Wobj:=Wobj_Part_0;
        Movel Tr_meulage_bavure_63,VitesseRapide,Z0,Tool \Wobj:=Wobj_Part_0;
        Movel Tr_meulage_bavure_64,VitesseRapide,Z0,Tool \Wobj:=Wobj_Part_0;
        Movel Tr_meulage_bavure_65,VitesseRapide,Z0,Tool \Wobj:=Wobj_Part_0;
        Movel Tr_meulage_bavure_66,VitesseRapide,Z0,Tool \Wobj:=Wobj_Part_0;
        Movel Tr_meulage_bavure_67,VitesseRapide,Z0,Tool \Wobj:=Wobj_Part_0;
        Movel Tr_meulage_bavure_68,VitesseRapide,Z0,Tool \Wobj:=Wobj_Part_0;
        Movel Tr_meulage_bavure_69,VitesseRapide,Z0,Tool \Wobj:=Wobj_Part_0;
        Movel Tr_meulage_bavure_70,VitesseRapide,Z0,Tool \Wobj:=Wobj_Part_0;
        Movel Tr_meulage_bavure_71,VitesseRapide,Z0,Tool \Wobj:=Wobj_Part_0;
        Movel Tr_meulage_bavure_72,VitesseRapide,Z0,Tool \Wobj:=Wobj_Part_0;
        Movel Tr_meulage_bavure_73,VitesseRapide,Z0,Tool \Wobj:=Wobj_Part_0;
        Movel Tr_meulage_bavure_74,VitesseRapide,Z0,Tool \Wobj:=Wobj_Part_0;
        Movel Tr_meulage_bavure_75,VitesseRapide,Z0,Tool \Wobj:=Wobj_Part_0;
        Movel Tr_meulage_bavure_76,VitesseRapide,Z0,Tool \Wobj:=Wobj_Part_0;
        Movel Tr_meulage_bavure_77,VitesseRapide,Z0,Tool \Wobj:=Wobj_Part_0;
        Movel Tr_meulage_bavure_78,VitesseRapide,Z0,Tool \Wobj:=Wobj_Part_0;
        Movel Tr_meulage_bavure_79,VitesseRapide,Z0,Tool \Wobj:=Wobj_Part_0;
        Movel Tr_meulage_bavure_80,VitesseRapide,Z0,Tool \Wobj:=Wobj_Part_0;
        Movel Tr_meulage_bavure_81,VitesseRapide,Z0,Tool \Wobj:=Wobj_Part_0;
        Movel Tr_meulage_bavure_82,VitesseRapide,Z0,Tool \Wobj:=Wobj_Part_0;
        Movel Tr_meulage_bavure_83,VitesseRapide,Z0,Tool \Wobj:=Wobj_Part_0;
        Movel Tr_meulage_bavure_84,VitesseRapide,Z0,Tool \Wobj:=Wobj_Part_0;
        Movel Tr_meulage_bavure_85,VitesseRapide,Z0,Tool \Wobj:=Wobj_Part_0;
        Movel Tr_meulage_bavure_86,VitesseRapide,Z0,Tool \Wobj:=Wobj_Part_0;
        Movel Tr_meulage_bavure_87,VitesseRapide,Z0,Tool \Wobj:=Wobj_Part_0;
        Movel Tr_meulage_bavure_88,VitesseRapide,Z0,Tool \Wobj:=Wobj_Part_0;
        Movel Tr_meulage_bavure_89,VitesseRapide,Z0,Tool \Wobj:=Wobj_Part_0;
        Movel Tr_meulage_bavure_90,VitesseRapide,Z0,Tool \Wobj:=Wobj_Part_0;
        Movel Tr_meulage_bavure_91,VitesseRapide,Z0,Tool \Wobj:=Wobj_Part_0;
        Movel Tr_meulage_bavure_92,VitesseRapide,Z0,Tool \Wobj:=Wobj_Part_0;
        Movel Tr_meulage_bavure_93,VitesseRapide,Z0,Tool \Wobj:=Wobj_Part_0;
        Movel Tr_meulage_bavure_94,VitesseRapide,Z0,Tool \Wobj:=Wobj_Part_0;
        Movel Tr_meulage_bavure_95,VitesseRapide,Z0,Tool \Wobj:=Wobj_Part_0;
        Movel Tr_meulage_bavure_96,VitesseRapide,Z0,Tool \Wobj:=Wobj_Part_0;
        Movel Tr_meulage_bavure_97,VitesseRapide,Z0,Tool \Wobj:=Wobj_Part_0;
        Movel Tr_meulage_bavure_98,VitesseRapide,Z0,Tool \Wobj:=Wobj_Part_0;
        Movel Tr_meulage_bavure_99,VitesseRapide,Z0,Tool \Wobj:=Wobj_Part_0;
        Movel Tr_meulage_bavure_100,VitesseRapide,Z0,Tool \Wobj:=Wobj_Part_0;
        Movel Tr_meulage_bavure_101,VitesseRapide,Z0,Tool \Wobj:=Wobj_Part_0;
        Movel Tr_meulage_bavure_102,VitesseRapide,Z0,Tool \Wobj:=Wobj_Part_0;
        Movel Tr_meulage_bavure_103,VitesseRapide,Z0,Tool \Wobj:=Wobj_Part_0;
        Movel Tr_meulage_bavure_104,VitesseRapide,Z0,Tool \Wobj:=Wobj_Part_0;
        Movel Tr_meulage_bavure_105,VitesseRapide,Z0,Tool \Wobj:=Wobj_Part_0;
        Movel Tr_meulage_bavure_106,VitesseRapide,Z0,Tool \Wobj:=Wobj_Part_0;
        Movel Tr_meulage_bavure_107,VitesseRapide,Z0,Tool \Wobj:=Wobj_Part_0;
        Movel Tr_meulage_bavure_108,VitesseRapide,Z0,Tool \Wobj:=Wobj_Part_0;
        Movel Tr_meulage_bavure_109,VitesseRapide,Z0,Tool \Wobj:=Wobj_Part_0;
        Movel Tr_meulage_bavure_110,VitesseRapide,Z0,Tool \Wobj:=Wobj_Part_0;
        Movel Tr_meulage_bavure_111,VitesseRapide,Z0,Tool \Wobj:=Wobj_Part_0;
        Movel Tr_meulage_bavure_112,VitesseRapide,Z0,Tool \Wobj:=Wobj_Part_0;
        Movel Tr_meulage_bavure_113,VitesseRapide,Z0,Tool \Wobj:=Wobj_Part_0;
        Movel Tr_meulage_bavure_114,VitesseRapide,Z0,Tool \Wobj:=Wobj_Part_0;
        Movel Tr_meulage_bavure_115,VitesseRapide,Z0,Tool \Wobj:=Wobj_Part_0;
        Movel Tr_meulage_bavure_116,VitesseRapide,Z0,Tool \Wobj:=Wobj_Part_0;
        Movel Tr_meulage_bavure_117,VitesseRapide,Z0,Tool \Wobj:=Wobj_Part_0;
        Movel Tr_meulage_bavure_118,VitesseRapide,Z0,Tool \Wobj:=Wobj_Part_0;
        Movel Tr_meulage_bavure_119,VitesseRapide,Z0,Tool \Wobj:=Wobj_Part_0;
        Movel Tr_meulage_bavure_120,VitesseRapide,Z0,Tool \Wobj:=Wobj_Part_0;
        Movel Tr_meulage_bavure_121,VitesseRapide,Z0,Tool \Wobj:=Wobj_Part_0;
        Movel Tr_meulage_bavure_122,VitesseRapide,Z0,Tool \Wobj:=Wobj_Part_0;
        Movel Tr_meulage_bavure_123,VitesseRapide,Z0,Tool \Wobj:=Wobj_Part_0;
        Movel Tr_meulage_bavure_124,VitesseRapide,Z0,Tool \Wobj:=Wobj_Part_0;
        Movel Tr_meulage_bavure_125,VitesseRapide,Z0,Tool \Wobj:=Wobj_Part_0;
        Movel Tr_meulage_bavure_126,VitesseRapide,Z0,Tool \Wobj:=Wobj_Part_0;
        Movel Tr_meulage_bavure_127,VitesseRapide,Z0,Tool \Wobj:=Wobj_Part_0;
        Movel Tr_meulage_bavure_128,VitesseRapide,Z0,Tool \Wobj:=Wobj_Part_0;
        Movel Tr_meulage_bavure_129,VitesseRapide,Z0,Tool \Wobj:=Wobj_Part_0;
        Movel Tr_meulage_bavure_130,VitesseRapide,Z0,Tool \Wobj:=Wobj_Part_0;
        Movel Tr_meulage_bavure_131,VitesseRapide,Z0,Tool \Wobj:=Wobj_Part_0;
        Movel Tr_meulage_bavure_132,VitesseRapide,Z0,Tool \Wobj:=Wobj_Part_0;
        Movel Tr_meulage_bavure_133,VitesseRapide,Z0,Tool \Wobj:=Wobj_Part_0;
        Movel Tr_meulage_bavure_134,VitesseRapide,Z0,Tool \Wobj:=Wobj_Part_0;
        Movel Tr_meulage_bavure_135,VitesseRapide,Z0,Tool \Wobj:=Wobj_Part_0;
        Movel Tr_meulage_bavure_136,VitesseRapide,Z0,Tool \Wobj:=Wobj_Part_0;
        Movel Tr_meulage_bavure_137,VitesseRapide,Z0,Tool \Wobj:=Wobj_Part_0;
        Movel Tr_meulage_bavure_138,VitesseRapide,Z0,Tool \Wobj:=Wobj_Part_0;
        Movel Tr_meulage_bavure_139,VitesseRapide,Z0,Tool \Wobj:=Wobj_Part_0;
        Movel Tr_meulage_bavure_140,VitesseRapide,Z0,Tool \Wobj:=Wobj_Part_0;
        Movel Tr_meulage_bavure_141,VitesseRapide,Z0,Tool \Wobj:=Wobj_Part_0;
        Movel Tr_meulage_bavure_142,VitesseRapide,Z0,Tool \Wobj:=Wobj_Part_0;
        Movel Tr_meulage_bavure_143,VitesseRapide,Z0,Tool \Wobj:=Wobj_Part_0;
        Movel Tr_meulage_bavure_144,VitesseRapide,Z0,Tool \Wobj:=Wobj_Part_0;
        Movel Tr_meulage_bavure_145,VitesseRapide,Z0,Tool \Wobj:=Wobj_Part_0;
        Movel Tr_meulage_bavure_146,VitesseRapide,Z0,Tool \Wobj:=Wobj_Part_0;
        Movel Tr_meulage_bavure_147,VitesseRapide,Z0,Tool \Wobj:=Wobj_Part_0;
        Movel Tr_meulage_bavure_148,VitesseRapide,Z0,Tool \Wobj:=Wobj_Part_0;
        Movel Tr_meulage_bavure_149,VitesseRapide,Z0,Tool \Wobj:=Wobj_Part_0;
        Movel Tr_meulage_bavure_150,VitesseRapide,Z0,Tool \Wobj:=Wobj_Part_0;
        Movel Tr_meulage_bavure_151,VitesseRapide,Z0,Tool \Wobj:=Wobj_Part_0;
        Movel Tr_meulage_bavure_152,VitesseRapide,Z0,Tool \Wobj:=Wobj_Part_0;
        Movel Tr_meulage_bavure_153,VitesseRapide,Z0,Tool \Wobj:=Wobj_Part_0;
        Movel Tr_meulage_bavure_154,VitesseRapide,Z0,Tool \Wobj:=Wobj_Part_0;
        Movel Tr_meulage_bavure_155,VitesseRapide,Z0,Tool \Wobj:=Wobj_Part_0;
        Movel Tr_meulage_bavure_156,VitesseRapide,Z0,Tool \Wobj:=Wobj_Part_0;
        Movel Tr_meulage_bavure_157,VitesseRapide,Z0,Tool \Wobj:=Wobj_Part_0;
        Movel Tr_meulage_bavure_158,VitesseRapide,Z0,Tool \Wobj:=Wobj_Part_0;
        Movel Tr_meulage_bavure_159,VitesseRapide,Z0,Tool \Wobj:=Wobj_Part_0;
        Movel Tr_meulage_bavure_160,VitesseRapide,Z0,Tool \Wobj:=Wobj_Part_0;
        Movel Tr_meulage_bavure_161,VitesseRapide,Z0,Tool \Wobj:=Wobj_Part_0;
        Movel Tr_meulage_bavure_162,VitesseRapide,Z0,Tool \Wobj:=Wobj_Part_0;
        Movel Tr_meulage_bavure_163,VitesseRapide,Z0,Tool \Wobj:=Wobj_Part_0;
        Movel Tr_meulage_bavure_164,VitesseRapide,Z0,Tool \Wobj:=Wobj_Part_0;
        Movel Tr_meulage_bavure_165,VitesseRapide,Z0,Tool \Wobj:=Wobj_Part_0;
        Movel Tr_meulage_bavure_166,VitesseRapide,Z0,Tool \Wobj:=Wobj_Part_0;
        Movel Tr_meulage_bavure_167,VitesseRapide,Z0,Tool \Wobj:=Wobj_Part_0;
        Movel Tr_meulage_bavure_168,VitesseRapide,Z0,Tool \Wobj:=Wobj_Part_0;
        Movel Tr_meulage_bavure_169,VitesseRapide,Z0,Tool \Wobj:=Wobj_Part_0;
        Movel Tr_meulage_bavure_170,VitesseRapide,Z0,Tool \Wobj:=Wobj_Part_0;
        Movel Tr_meulage_bavure_171,VitesseRapide,Z0,Tool \Wobj:=Wobj_Part_0;
        Movel Tr_meulage_bavure_172,VitesseRapide,Z0,Tool \Wobj:=Wobj_Part_0;
        Movel Tr_meulage_bavure_173,VitesseRapide,Z0,Tool \Wobj:=Wobj_Part_0;
        Movel Tr_meulage_bavure_174,VitesseRapide,Z0,Tool \Wobj:=Wobj_Part_0;
        Movel Tr_meulage_bavure_175,VitesseRapide,Z0,Tool \Wobj:=Wobj_Part_0;
        Movel Tr_meulage_bavure_176,VitesseRapide,Z0,Tool \Wobj:=Wobj_Part_0;
        Movel Tr_meulage_bavure_177,VitesseRapide,Z0,Tool \Wobj:=Wobj_Part_0;
        Movel Tr_meulage_bavure_178,VitesseRapide,Z0,Tool \Wobj:=Wobj_Part_0;
        Movel Tr_meulage_bavure_179,VitesseRapide,Z0,Tool \Wobj:=Wobj_Part_0;
        Movel Tr_meulage_bavure_180,VitesseRapide,Z0,Tool \Wobj:=Wobj_Part_0;
        Movel Tr_meulage_bavure_181,VitesseRapide,Z0,Tool \Wobj:=Wobj_Part_0;
        Movel Tr_meulage_bavure_182,VitesseRapide,Z0,Tool \Wobj:=Wobj_Part_0;
        Movel Tr_meulage_bavure_183,VitesseRapide,Z0,Tool \Wobj:=Wobj_Part_0;
        Movel Tr_meulage_bavure_184,VitesseRapide,Z0,Tool \Wobj:=Wobj_Part_0;
        Movel Tr_meulage_bavure_185,VitesseRapide,Z0,Tool \Wobj:=Wobj_Part_0;
        Movel Tr_meulage_bavure_186,VitesseRapide,Z0,Tool \Wobj:=Wobj_Part_0;
        Movel Tr_meulage_bavure_187,VitesseRapide,Z0,Tool \Wobj:=Wobj_Part_0;
        Movel Tr_meulage_bavure_188,VitesseRapide,Z0,Tool \Wobj:=Wobj_Part_0;
        Movel Tr_meulage_bavure_189,VitesseRapide,Z0,Tool \Wobj:=Wobj_Part_0;
        Movel Tr_meulage_bavure_190,VitesseRapide,Z0,Tool \Wobj:=Wobj_Part_0;
        Movel Tr_meulage_bavure_191,VitesseRapide,Z0,Tool \Wobj:=Wobj_Part_0;
        Movel Tr_meulage_bavure_192,VitesseRapide,Z0,Tool \Wobj:=Wobj_Part_0;
        Movel Tr_meulage_bavure_193,VitesseRapide,Z0,Tool \Wobj:=Wobj_Part_0;
        Movel Tr_meulage_bavure_194,VitesseRapide,Z0,Tool \Wobj:=Wobj_Part_0;
        Movel Tr_meulage_bavure_195,VitesseRapide,Z0,Tool \Wobj:=Wobj_Part_0;
        Movel Tr_meulage_bavure_196,VitesseRapide,Z0,Tool \Wobj:=Wobj_Part_0;
        Movel Tr_meulage_bavure_197,VitesseRapide,Z0,Tool \Wobj:=Wobj_Part_0;
        Movel Tr_meulage_bavure_198,VitesseRapide,Z0,Tool \Wobj:=Wobj_Part_0;
        Movel Tr_meulage_bavure_199,VitesseRapide,Z0,Tool \Wobj:=Wobj_Part_0;
        Movel Tr_meulage_bavure_200,VitesseRapide,Z0,Tool \Wobj:=Wobj_Part_0;
        Movel Tr_meulage_bavure_201,VitesseRapide,Z0,Tool \Wobj:=Wobj_Part_0;
        Movel Tr_meulage_bavure_202,VitesseRapide,Z0,Tool \Wobj:=Wobj_Part_0;
        Movel Tr_meulage_bavure_203,VitesseRapide,Z0,Tool \Wobj:=Wobj_Part_0;
        Movel Tr_meulage_bavure_204,VitesseRapide,Z0,Tool \Wobj:=Wobj_Part_0;
        Movel Tr_meulage_bavure_205,VitesseRapide,Z0,Tool \Wobj:=Wobj_Part_0;
        Movel Tr_meulage_bavure_206,VitesseRapide,Z0,Tool \Wobj:=Wobj_Part_0;
        Movel Tr_meulage_bavure_207,VitesseRapide,Z0,Tool \Wobj:=Wobj_Part_0;
        Movel Tr_meulage_bavure_208,VitesseRapide,Z0,Tool \Wobj:=Wobj_Part_0;
        Movel Tr_meulage_bavure_209,VitesseRapide,Z0,Tool \Wobj:=Wobj_Part_0;
        Movel Tr_meulage_bavure_210,VitesseRapide,Z0,Tool \Wobj:=Wobj_Part_0;
        Movel Tr_meulage_bavure_211,VitesseRapide,Z0,Tool \Wobj:=Wobj_Part_0;
        Movel Tr_meulage_bavure_212,VitesseRapide,Z0,Tool \Wobj:=Wobj_Part_0;
        Movel Tr_meulage_bavure_213,VitesseRapide,Z0,Tool \Wobj:=Wobj_Part_0;
        Movel Tr_meulage_bavure_214,VitesseRapide,Z0,Tool \Wobj:=Wobj_Part_0;
        Movel Tr_meulage_bavure_215,VitesseRapide,Z0,Tool \Wobj:=Wobj_Part_0;
        Movel Tr_meulage_bavure_216,VitesseRapide,Z0,Tool \Wobj:=Wobj_Part_0;
        Movel Tr_meulage_bavure_217,VitesseRapide,Z0,Tool \Wobj:=Wobj_Part_0;
        Movel Tr_meulage_bavure_218,VitesseRapide,Z0,Tool \Wobj:=Wobj_Part_0;
        Movel Tr_meulage_bavure_219,VitesseRapide,Z0,Tool \Wobj:=Wobj_Part_0;
        Movel Tr_meulage_bavure_220,VitesseRapide,Z0,Tool \Wobj:=Wobj_Part_0;
        Movel Tr_meulage_bavure_221,VitesseRapide,Z0,Tool \Wobj:=Wobj_Part_0;
        Movel Tr_meulage_bavure_222,VitesseRapide,Z0,Tool \Wobj:=Wobj_Part_0;
        Movel Tr_meulage_bavure_223,VitesseRapide,Z0,Tool \Wobj:=Wobj_Part_0;
        Movel Tr_meulage_bavure_224,VitesseRapide,Z0,Tool \Wobj:=Wobj_Part_0;
        Movel Tr_meulage_bavure_225,VitesseRapide,Z0,Tool \Wobj:=Wobj_Part_0;
        Movel Tr_meulage_bavure_226,VitesseRapide,Z0,Tool \Wobj:=Wobj_Part_0;
        Movel Tr_meulage_bavure_227,VitesseRapide,Z0,Tool \Wobj:=Wobj_Part_0;
        Movel Tr_meulage_bavure_228,VitesseRapide,Z0,Tool \Wobj:=Wobj_Part_0;
        Movel Tr_meulage_bavure_229,VitesseRapide,Z0,Tool \Wobj:=Wobj_Part_0;
        Movel Tr_meulage_bavure_230,VitesseRapide,Z0,Tool \Wobj:=Wobj_Part_0;
        Movel Tr_meulage_bavure_231,VitesseRapide,Z0,Tool \Wobj:=Wobj_Part_0;
        Movel Tr_meulage_bavure_232,VitesseRapide,Z0,Tool \Wobj:=Wobj_Part_0;
        Movel Tr_meulage_bavure_233,VitesseRapide,Z0,Tool \Wobj:=Wobj_Part_0;
        Movel Tr_meulage_bavure_234,VitesseRapide,Z0,Tool \Wobj:=Wobj_Part_0;
        Movel Tr_meulage_bavure_235,VitesseRapide,Z0,Tool \Wobj:=Wobj_Part_0;
        Movel Tr_meulage_bavure_236,VitesseRapide,Z0,Tool \Wobj:=Wobj_Part_0;
        Movel Tr_meulage_bavure_237,VitesseRapide,Z0,Tool \Wobj:=Wobj_Part_0;
        Movel Tr_meulage_bavure_238,VitesseRapide,Z0,Tool \Wobj:=Wobj_Part_0;
        Movel Tr_meulage_bavure_239,VitesseRapide,Z0,Tool \Wobj:=Wobj_Part_0;
        Movel Tr_meulage_bavure_240,VitesseRapide,Z0,Tool \Wobj:=Wobj_Part_0;
        Movel Tr_meulage_bavure_241,VitesseRapide,Z0,Tool \Wobj:=Wobj_Part_0;
        Movel Tr_meulage_bavure_242,VitesseRapide,Z0,Tool \Wobj:=Wobj_Part_0;
        Movel Tr_meulage_bavure_243,VitesseRapide,Z0,Tool \Wobj:=Wobj_Part_0;
        Movel Tr_meulage_bavure_244,VitesseRapide,Z0,Tool \Wobj:=Wobj_Part_0;
        Movel Tr_meulage_bavure_245,VitesseRapide,Z0,Tool \Wobj:=Wobj_Part_0;
        Movel Tr_meulage_bavure_246,VitesseRapide,Z0,Tool \Wobj:=Wobj_Part_0;
        Movel Tr_meulage_bavure_247,VitesseRapide,Z0,Tool \Wobj:=Wobj_Part_0;
        Movel Tr_meulage_bavure_248,VitesseRapide,Z0,Tool \Wobj:=Wobj_Part_0;
        Movel Tr_meulage_bavure_249,VitesseRapide,Z0,Tool \Wobj:=Wobj_Part_0;
        Movel Tr_meulage_bavure_250,VitesseRapide,Z0,Tool \Wobj:=Wobj_Part_0;
        Movel Tr_meulage_bavure_251,VitesseRapide,Z0,Tool \Wobj:=Wobj_Part_0;
        Movel Tr_meulage_bavure_252,VitesseRapide,Z0,Tool \Wobj:=Wobj_Part_0;
        Movel Tr_meulage_bavure_253,VitesseRapide,Z0,Tool \Wobj:=Wobj_Part_0;
        Movel Tr_meulage_bavure_254,VitesseRapide,Z0,Tool \Wobj:=Wobj_Part_0;
        Movel Tr_meulage_bavure_255,VitesseRapide,Z0,Tool \Wobj:=Wobj_Part_0;
        Movel Tr_meulage_bavure_256,VitesseRapide,Z0,Tool \Wobj:=Wobj_Part_0;
        Movel Tr_meulage_bavure_257,VitesseRapide,Z0,Tool \Wobj:=Wobj_Part_0;
        Movel Tr_meulage_bavure_258,VitesseRapide,Z0,Tool \Wobj:=Wobj_Part_0;
        Movel Tr_meulage_bavure_259,VitesseRapide,Z0,Tool \Wobj:=Wobj_Part_0;
        Movel Tr_meulage_bavure_260,VitesseRapide,Z0,Tool \Wobj:=Wobj_Part_0;
        Movel Tr_meulage_bavure_261,VitesseRapide,Z0,Tool \Wobj:=Wobj_Part_0;
        Movel Tr_meulage_bavure_262,VitesseRapide,Z0,Tool \Wobj:=Wobj_Part_0;
        Movel Tr_meulage_bavure_263,VitesseRapide,Z0,Tool \Wobj:=Wobj_Part_0;
        Movel Tr_meulage_bavure_264,VitesseRapide,Z0,Tool \Wobj:=Wobj_Part_0;
        Movel Tr_meulage_bavure_265,VitesseRapide,Z0,Tool \Wobj:=Wobj_Part_0;
        Movel Tr_meulage_bavure_266,VitesseRapide,Z0,Tool \Wobj:=Wobj_Part_0;
        Movel Tr_meulage_bavure_267,VitesseRapide,Z0,Tool \Wobj:=Wobj_Part_0;
        Movel Tr_meulage_bavure_268,VitesseRapide,Z0,Tool \Wobj:=Wobj_Part_0;
        Movel Tr_meulage_bavure_269,VitesseRapide,Z0,Tool \Wobj:=Wobj_Part_0;
        Movel Tr_meulage_bavure_270,VitesseRapide,Z0,Tool \Wobj:=Wobj_Part_0;
        Movel Tr_meulage_bavure_271,VitesseRapide,Z0,Tool \Wobj:=Wobj_Part_0;
        Movel Tr_meulage_bavure_272,VitesseRapide,Z0,Tool \Wobj:=Wobj_Part_0;
        Movel Tr_meulage_bavure_273,VitesseRapide,Z0,Tool \Wobj:=Wobj_Part_0;
        Movel Tr_meulage_bavure_274,VitesseRapide,Z0,Tool \Wobj:=Wobj_Part_0;
        Movel Tr_meulage_bavure_275,VitesseRapide,Z0,Tool \Wobj:=Wobj_Part_0;
        Movel Tr_meulage_bavure_276,VitesseRapide,Z0,Tool \Wobj:=Wobj_Part_0;
        Movel Tr_meulage_bavure_277,VitesseRapide,Z0,Tool \Wobj:=Wobj_Part_0;
        Movel Tr_meulage_bavure_278,VitesseRapide,Z0,Tool \Wobj:=Wobj_Part_0;
        Movel Tr_meulage_bavure_279,VitesseRapide,Z0,Tool \Wobj:=Wobj_Part_0;
        Movel Tr_meulage_bavure_280,VitesseRapide,Z0,Tool \Wobj:=Wobj_Part_0;
        Movel Tr_meulage_bavure_281,VitesseRapide,Z0,Tool \Wobj:=Wobj_Part_0;
        Movel Tr_meulage_bavure_282,VitesseRapide,Z0,Tool \Wobj:=Wobj_Part_0;
        Movel Tr_meulage_bavure_283,VitesseRapide,Z0,Tool \Wobj:=Wobj_Part_0;
        Movel Tr_meulage_bavure_284,VitesseRapide,Z0,Tool \Wobj:=Wobj_Part_0;
        Movel Tr_meulage_bavure_285,VitesseRapide,Z0,Tool \Wobj:=Wobj_Part_0;
        Movel Tr_meulage_bavure_286,VitesseRapide,Z0,Tool \Wobj:=Wobj_Part_0;
        Movel Tr_meulage_bavure_287,VitesseRapide,Z0,Tool \Wobj:=Wobj_Part_0;
        Movel Tr_meulage_bavure_288,VitesseRapide,Z0,Tool \Wobj:=Wobj_Part_0;
        Movel Tr_meulage_bavure_289,VitesseRapide,Z0,Tool \Wobj:=Wobj_Part_0;
        Movel Tr_meulage_bavure_290,VitesseRapide,Z0,Tool \Wobj:=Wobj_Part_0;
        Movel Tr_meulage_bavure_291,VitesseRapide,Z0,Tool \Wobj:=Wobj_Part_0;
        Movel Tr_meulage_bavure_292,VitesseRapide,Z0,Tool \Wobj:=Wobj_Part_0;
        Movel Tr_meulage_bavure_293,VitesseRapide,Z0,Tool \Wobj:=Wobj_Part_0;
        Movel Tr_meulage_bavure_294,VitesseRapide,Z0,Tool \Wobj:=Wobj_Part_0;
        Movel Tr_meulage_bavure_295,VitesseRapide,Z0,Tool \Wobj:=Wobj_Part_0;
        Movel Tr_meulage_bavure_296,VitesseRapide,Z0,Tool \Wobj:=Wobj_Part_0;
        Movel Tr_meulage_bavure_297,VitesseRapide,Z0,Tool \Wobj:=Wobj_Part_0;
        Movel Tr_meulage_bavure_298,VitesseRapide,Z0,Tool \Wobj:=Wobj_Part_0;
        Movel Tr_meulage_bavure_299,VitesseRapide,Z0,Tool \Wobj:=Wobj_Part_0;
        Movel Tr_meulage_bavure_300,VitesseRapide,Z0,Tool \Wobj:=Wobj_Part_0;
        Movel Tr_meulage_bavure_301,VitesseRapide,Z0,Tool \Wobj:=Wobj_Part_0;
        Movel Tr_meulage_bavure_302,VitesseRapide,Z0,Tool \Wobj:=Wobj_Part_0;
        Movel Tr_meulage_bavure_303,VitesseRapide,Z0,Tool \Wobj:=Wobj_Part_0;
        Movel Tr_meulage_bavure_304,VitesseRapide,Z0,Tool \Wobj:=Wobj_Part_0;
        Movel Tr_meulage_bavure_305,VitesseRapide,Z0,Tool \Wobj:=Wobj_Part_0;
        Movel Tr_meulage_bavure_306,VitesseRapide,Z0,Tool \Wobj:=Wobj_Part_0;
        Movel Tr_meulage_bavure_307,VitesseRapide,Z0,Tool \Wobj:=Wobj_Part_0;
        Movel Tr_meulage_bavure_308,VitesseRapide,Z0,Tool \Wobj:=Wobj_Part_0;
        Movel Tr_meulage_bavure_309,VitesseRapide,Z0,Tool \Wobj:=Wobj_Part_0;
        Movel Tr_meulage_bavure_310,VitesseRapide,Z0,Tool \Wobj:=Wobj_Part_0;
        Movel Tr_meulage_bavure_311,VitesseRapide,Z0,Tool \Wobj:=Wobj_Part_0;
        Movel Tr_meulage_bavure_312,VitesseRapide,Z0,Tool \Wobj:=Wobj_Part_0;
        Movel Tr_meulage_bavure_313,VitesseRapide,Z0,Tool \Wobj:=Wobj_Part_0;
        Movel Tr_meulage_bavure_314,VitesseRapide,Z0,Tool \Wobj:=Wobj_Part_0;
        Movel Tr_meulage_bavure_315,VitesseRapide,Z0,Tool \Wobj:=Wobj_Part_0;
        Movel Tr_meulage_bavure_316,VitesseRapide,Z0,Tool \Wobj:=Wobj_Part_0;
        Movel Tr_meulage_bavure_317,VitesseRapide,Z0,Tool \Wobj:=Wobj_Part_0;
        Movel Tr_meulage_bavure_318,VitesseRapide,Z0,Tool \Wobj:=Wobj_Part_0;
        Movel Tr_meulage_bavure_319,VitesseRapide,Z0,Tool \Wobj:=Wobj_Part_0;
        Movel Tr_meulage_bavure_320,VitesseRapide,Z0,Tool \Wobj:=Wobj_Part_0;
        Movel Tr_meulage_bavure_321,VitesseRapide,Z0,Tool \Wobj:=Wobj_Part_0;
        Movel Tr_meulage_bavure_322,VitesseRapide,Z0,Tool \Wobj:=Wobj_Part_0;
        Movel Tr_meulage_bavure_323,VitesseRapide,Z0,Tool \Wobj:=Wobj_Part_0;
        Movel Tr_meulage_bavure_324,VitesseRapide,Z0,Tool \Wobj:=Wobj_Part_0;
        Movel Tr_meulage_bavure_325,VitesseRapide,Z0,Tool \Wobj:=Wobj_Part_0;
        Movel Tr_meulage_bavure_326,VitesseRapide,Z0,Tool \Wobj:=Wobj_Part_0;
        Movel Tr_meulage_bavure_327,VitesseRapide,Z0,Tool \Wobj:=Wobj_Part_0;
        Movel Tr_meulage_bavure_328,VitesseRapide,Z0,Tool \Wobj:=Wobj_Part_0;
        Movel Tr_meulage_bavure_329,VitesseRapide,Z0,Tool \Wobj:=Wobj_Part_0;
        Movel Tr_meulage_bavure_330,VitesseRapide,Z0,Tool \Wobj:=Wobj_Part_0;
        Movel Tr_meulage_bavure_331,VitesseRapide,Z0,Tool \Wobj:=Wobj_Part_0;
        Movel Tr_meulage_bavure_332,VitesseRapide,Z0,Tool \Wobj:=Wobj_Part_0;
        Movel Tr_meulage_bavure_333,VitesseRapide,Z0,Tool \Wobj:=Wobj_Part_0;
        Movel Tr_meulage_bavure_334,VitesseRapide,Z0,Tool \Wobj:=Wobj_Part_0;
        Movel Tr_meulage_bavure_335,VitesseRapide,Z0,Tool \Wobj:=Wobj_Part_0;
        Movel Tr_meulage_bavure_336,VitesseRapide,Z0,Tool \Wobj:=Wobj_Part_0;
        Movel Tr_meulage_bavure_337,VitesseRapide,Z0,Tool \Wobj:=Wobj_Part_0;
        Movel Tr_meulage_bavure_338,VitesseRapide,Z0,Tool \Wobj:=Wobj_Part_0;
        Movel Tr_meulage_bavure_339,VitesseRapide,Z0,Tool \Wobj:=Wobj_Part_0;
        Movel Tr_meulage_bavure_340,VitesseRapide,Z0,Tool \Wobj:=Wobj_Part_0;
        Movel Tr_meulage_bavure_341,VitesseRapide,Z0,Tool \Wobj:=Wobj_Part_0;
        Movel Tr_meulage_bavure_342,VitesseRapide,Z0,Tool \Wobj:=Wobj_Part_0;
        Movel Tr_meulage_bavure_343,VitesseRapide,Z0,Tool \Wobj:=Wobj_Part_0;
        Movel Tr_meulage_bavure_344,VitesseRapide,Z0,Tool \Wobj:=Wobj_Part_0;
        Movel Tr_meulage_bavure_345,VitesseRapide,Z0,Tool \Wobj:=Wobj_Part_0;
        Movel Tr_meulage_bavure_346,VitesseRapide,Z0,Tool \Wobj:=Wobj_Part_0;
        Movel Tr_meulage_bavure_347,VitesseRapide,Z0,Tool \Wobj:=Wobj_Part_0;
        Movel Tr_meulage_bavure_348,VitesseRapide,Z0,Tool \Wobj:=Wobj_Part_0;
        Movel Tr_meulage_bavure_349,VitesseRapide,Z0,Tool \Wobj:=Wobj_Part_0;
        Movel Tr_meulage_bavure_350,VitesseRapide,Z0,Tool \Wobj:=Wobj_Part_0;
        Movel Tr_meulage_bavure_351,VitesseRapide,Z0,Tool \Wobj:=Wobj_Part_0;
        Movel Tr_meulage_bavure_352,VitesseRapide,Z0,Tool \Wobj:=Wobj_Part_0;
        Movel Tr_meulage_bavure_353,VitesseRapide,Z0,Tool \Wobj:=Wobj_Part_0;
        Movel Tr_meulage_bavure_354,VitesseRapide,Z0,Tool \Wobj:=Wobj_Part_0;
        Movel Tr_meulage_bavure_355,VitesseRapide,Z0,Tool \Wobj:=Wobj_Part_0;
        Movel Tr_meulage_bavure_356,VitesseRapide,Z0,Tool \Wobj:=Wobj_Part_0;
        Movel Tr_meulage_bavure_357,VitesseRapide,Z0,Tool \Wobj:=Wobj_Part_0;
        Movel Tr_meulage_bavure_358,VitesseRapide,Z0,Tool \Wobj:=Wobj_Part_0;
        Movel Tr_meulage_bavure_359,VitesseRapide,Z0,Tool \Wobj:=Wobj_Part_0;
        Movel Tr_meulage_bavure_360,VitesseRapide,Z0,Tool \Wobj:=Wobj_Part_0;
        Movel Tr_meulage_bavure_361,VitesseRapide,Z0,Tool \Wobj:=Wobj_Part_0;
        Movel Tr_meulage_bavure_362,VitesseRapide,Z0,Tool \Wobj:=Wobj_Part_0;
        Movel Tr_meulage_bavure_363,VitesseRapide,Z0,Tool \Wobj:=Wobj_Part_0;
        Movel Tr_meulage_bavure_364,VitesseRapide,Z0,Tool \Wobj:=Wobj_Part_0;
        Movel Tr_meulage_bavure_365,VitesseRapide,Z0,Tool \Wobj:=Wobj_Part_0;
        Movel Tr_meulage_bavure_366,VitesseRapide,Z0,Tool \Wobj:=Wobj_Part_0;
        Movel Tr_meulage_bavure_367,VitesseRapide,Z0,Tool \Wobj:=Wobj_Part_0;
        Movel Tr_meulage_bavure_368,VitesseRapide,Z0,Tool \Wobj:=Wobj_Part_0;
        Movel Tr_meulage_bavure_369,VitesseRapide,Z0,Tool \Wobj:=Wobj_Part_0;
        Movel Tr_meulage_bavure_370,VitesseRapide,Z0,Tool \Wobj:=Wobj_Part_0;
        Movel Tr_meulage_bavure_371,VitesseRapide,Z0,Tool \Wobj:=Wobj_Part_0;
        Movel Tr_meulage_bavure_372,VitesseRapide,Z0,Tool \Wobj:=Wobj_Part_0;
        Movel Tr_meulage_bavure_373,VitesseRapide,Z0,Tool \Wobj:=Wobj_Part_0;
        Movel Tr_meulage_bavure_374,VitesseRapide,Z0,Tool \Wobj:=Wobj_Part_0;
        Movel Tr_meulage_bavure_375,VitesseRapide,Z0,Tool \Wobj:=Wobj_Part_0;
        Movel Tr_meulage_bavure_376,VitesseRapide,Z0,Tool \Wobj:=Wobj_Part_0;
        Movel Tr_meulage_bavure_377,VitesseRapide,Z0,Tool \Wobj:=Wobj_Part_0;
        Movel Tr_meulage_bavure_378,VitesseRapide,Z0,Tool \Wobj:=Wobj_Part_0;
        Movel Tr_meulage_bavure_379,VitesseRapide,Z0,Tool \Wobj:=Wobj_Part_0;
        Movel Tr_meulage_bavure_380,VitesseRapide,Z0,Tool \Wobj:=Wobj_Part_0;
        Movel Tr_meulage_bavure_381,VitesseRapide,Z0,Tool \Wobj:=Wobj_Part_0;
        Movel Tr_meulage_bavure_382,VitesseRapide,Z0,Tool \Wobj:=Wobj_Part_0;
        Movel Tr_meulage_bavure_383,VitesseRapide,Z0,Tool \Wobj:=Wobj_Part_0;
        Movel Tr_meulage_bavure_384,VitesseRapide,Z0,Tool \Wobj:=Wobj_Part_0;
        Movel Tr_meulage_bavure_385,VitesseRapide,Z0,Tool \Wobj:=Wobj_Part_0;
        Movel Tr_meulage_bavure_386,VitesseRapide,Z0,Tool \Wobj:=Wobj_Part_0;
        Movel Tr_meulage_bavure_387,VitesseRapide,Z0,Tool \Wobj:=Wobj_Part_0;
        Movel Tr_meulage_bavure_388,VitesseRapide,Z0,Tool \Wobj:=Wobj_Part_0;
        Movel Tr_meulage_bavure_389,VitesseRapide,Z0,Tool \Wobj:=Wobj_Part_0;
        Movel Tr_meulage_bavure_390,VitesseRapide,Z0,Tool \Wobj:=Wobj_Part_0;
        Movel Tr_meulage_bavure_391,VitesseRapide,Z0,Tool \Wobj:=Wobj_Part_0;
        !
        !Degagement
        MoveL Reltool(Tr_meulage_bavure_391,0,0,-10),V100,Z0,Tool \Wobj:=Wobj_Part_0;
        MoveL Reltool(Tr_meulage_bavure_391,0,0,-100),V500,Z0,Tool \Wobj:=Wobj_Part_0;
        MoveJ Reltool(Tr_meulage_bavure_391,0,0,-200),V1000,Z0,Tool \Wobj:=Wobj_Part_0;


        Go_to_Meulage_Plan;
        !
        !

    ENDPROC

    !Trajectoire de depose de la piece
    LOCAL PROC DEPOSE()
        !
        stop;

        PEO;

        !
        !Approche
		MoveJ Reltool(PicKPosition,0,0,-200),V1000,Z0,Tool_Prehenseur1 \Wobj:=Wobj_vision;
		MoveL Reltool(PicKPosition,0,0,-100),V500,Z0,Tool_Prehenseur1 \Wobj:=Wobj_vision;
		MoveL Reltool(PicKPosition,0,0,-10),V200,Z0,Tool_Prehenseur1 \Wobj:=Wobj_vision;
		MoveL PicKPosition,V100,Fine,Tool_Prehenseur1 \Wobj:=Wobj_vision;

        !Fermeture pince
		Gripper_Open;
        !
		MoveL Reltool(PicKPosition,0,0,-200),V500,Z0,Tool_Prehenseur1 \Wobj:=Wobj_vision;

        !
        PEO;
        !

        !Gripper_Close;

        !
    ENDPROC

ENDMODULE
